{attribute 'qualified_only'}
VAR_GLOBAL
	Fixture1Input:FixtureInput;
	Fixture1Output:FixtureOutput;
	Fixture2Input:FixtureInput;
	Fixture2Output:FixtureOutput;
END_VAR

(* stored: Version 1.1.0.1, ProductVersion 3.1.4024.16
   GVL IO_1: Id {d33c385b-972c-4192-9b5b-190b0cd51b4b} *)
